// Mitsubishi GX Developer project: 小车运行控制   PLC: FX3U

PROGRAM MAIN
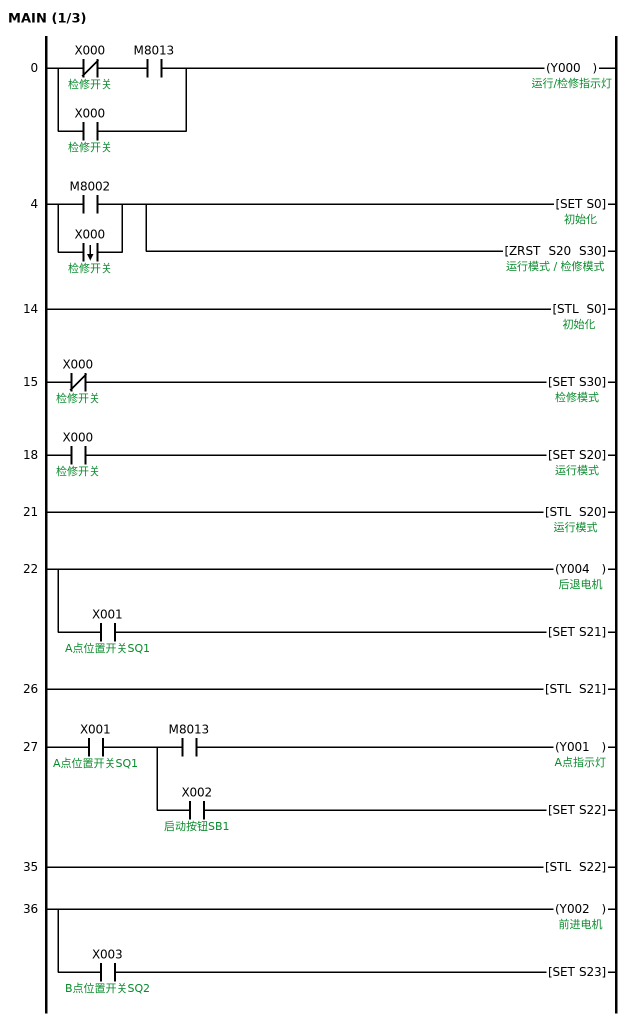
0     LDI     X000  ; 检修开关
      AND     M8013
      OR      X000  ; 检修开关
      OUT     Y000  ; 运行/检修指示灯
4     LD      M8002
      ORF     X000  ; 检修开关
      SET     S0  ; 初始化
      ZRST    S20 S30  ; 运行模式 / 检修模式
14    STL     S0
15    LDI     X000  ; 检修开关
      SET     S30  ; 检修模式
18    LD      X000  ; 检修开关
      SET     S20  ; 运行模式
21    STL     S20
22    OUT     Y004  ; 后退电机
      AND     X001  ; A点位置开关SQ1
      SET     S21
26    STL     S21
27    LD      X001  ; A点位置开关SQ1
      MPS
      AND     M8013
      OUT     Y001  ; A点指示灯
      MPP
      AND     X002  ; 启动按钮SB1
      SET     S22
35    STL     S22
36    OUT     Y002  ; 前进电机
      AND     X003  ; B点位置开关SQ2
      SET     S23
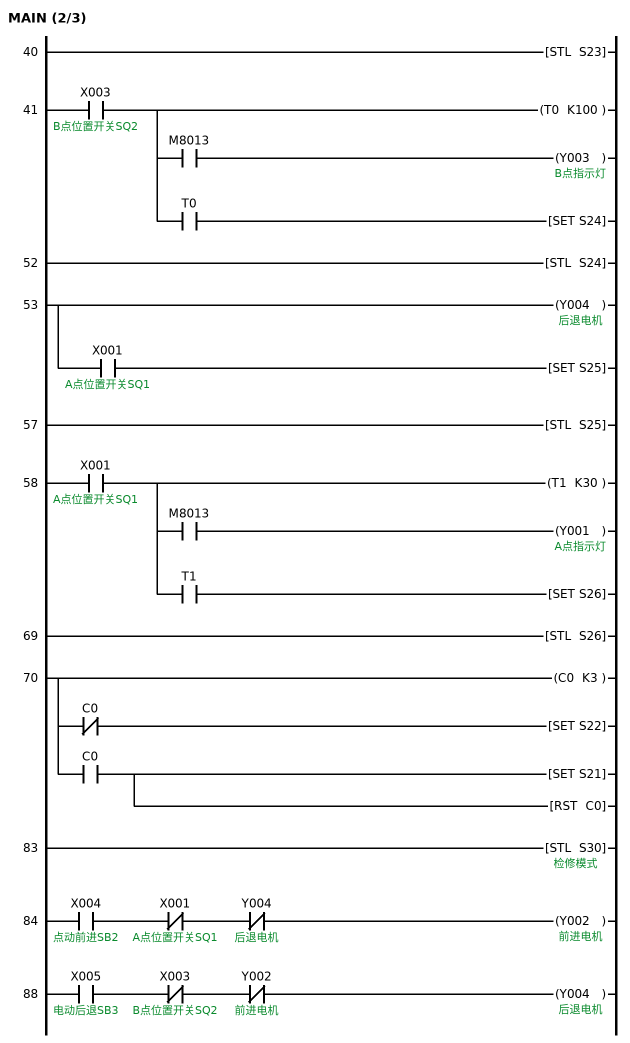
40    STL     S23
41    LD      X003  ; B点位置开关SQ2
      OUT     T0 K100
      MPS
      AND     M8013
      OUT     Y003  ; B点指示灯
      MPP
      AND     T0
      SET     S24
52    STL     S24
53    OUT     Y004  ; 后退电机
      AND     X001  ; A点位置开关SQ1
      SET     S25
57    STL     S25
58    LD      X001  ; A点位置开关SQ1
      OUT     T1 K30
      MPS
      AND     M8013
      OUT     Y001  ; A点指示灯
      MPP
      AND     T1
      SET     S26
69    STL     S26
70    OUT     C0 K3
      MPS
      ANI     C0
      SET     S22
      MPP
      AND     C0
      SET     S21
      RST     C0
83    STL     S30
84    LD      X004  ; 点动前进SB2
      ANI     X001  ; A点位置开关SQ1
      ANI     Y004  ; 后退电机
      OUT     Y002  ; 前进电机
88    LD      X005  ; 电动后退SB3
      ANI     X003  ; B点位置开关SQ2
      ANI     Y002  ; 前进电机
      OUT     Y004  ; 后退电机
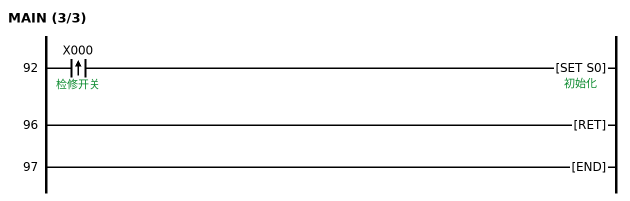
92    LDP     X000  ; 检修开关
      SET     S0  ; 初始化
96    RET
97    END
END_PROGRAM
